# EPICS substitutions: db/Beckhoff_1XXX/ecmcEKM1101.substitutions
file "ecmcEcSlave.template"
{
  pattern {}
          {}
}

file "ecmcEKM1101-DEV.template"
{
  pattern {}
          {}
}

file "ecmcEKM1101-ACC.template"
{
  pattern {CH_ID, LINR,    ESLO,            EOFF,   EGU,     PREC, LOW, LOLO, HIGH, HIHI, HYST, LLSV,       LSV,        HSV,        HHSV      }
          {X,     "SLOPE", 1,        0,      "g",     3,    0,   0,    0,    0,    0,    "NO_ALARM", "NO_ALARM", "NO_ALARM", "NO_ALARM"}
          {Y,     "SLOPE", 1,        0,      "g",     3,    0,   0,    0,    0,    0,    "NO_ALARM", "NO_ALARM", "NO_ALARM", "NO_ALARM"}
          {Z,     "SLOPE", 1,        0,      "g",     3,    0,   0,    0,    0,    0,    "NO_ALARM", "NO_ALARM", "NO_ALARM", "NO_ALARM"}
}

file "ecmcEKM1101-VOL.template"
{
  pattern {CH_ID, LINR,    ESLO,            EOFF,   EGU,     PREC, LOW, LOLO, HIGH, HIHI, HYST, LLSV,       LSV,        HSV,        HHSV      }
          {USIN,  "SLOPE", 2.3283064e-8,    0,      "V",     0,    0,   0,    0,    0,    0,    "NO_ALARM", "NO_ALARM", "NO_ALARM", "NO_ALARM"}
          {UPIN,  "SLOPE", 2.3283064e-8,    0,      "V",     0,    0,   0,    0,    0,    0,    "NO_ALARM", "NO_ALARM", "NO_ALARM", "NO_ALARM"}
          {UPOUT, "SLOPE", 2.3283064e-8,    0,      "V",     0,    0,   0,    0,    0,    0,    "NO_ALARM", "NO_ALARM", "NO_ALARM", "NO_ALARM"}
}
